FUNCTION_BLOCK plant
  (* Standard: 61499-2 *)
  (* Version 0.1, 2017-00-25, hpea485, UOA *)
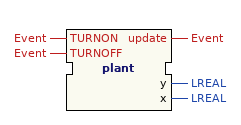
  EVENT_INPUT
    TURNON;
    TURNOFF;
  END_EVENT
  EVENT_OUTPUT
    update;
  END_EVENT
  VAR_OUTPUT
    y : LREAL;
    x : LREAL;
  END_VAR
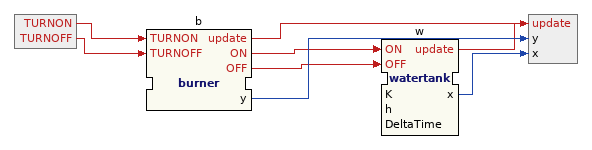
  FBS
    b : burner;
    w : watertank;
  END_FBS
  EVENT_CONNECTIONS
    TURNON TO b.TURNON;
    TURNOFF TO b.TURNOFF;
    b.update TO update;
    w.update TO update;
    b.ON TO w.ON;
    b.OFF TO w.OFF;
  END_CONNECTIONS
  DATA_CONNECTIONS
    b.y TO y;
    w.x TO x;
  END_CONNECTIONS
END_FUNCTION_BLOCK
